Yaskawa INFORM job: DROP01.JBI

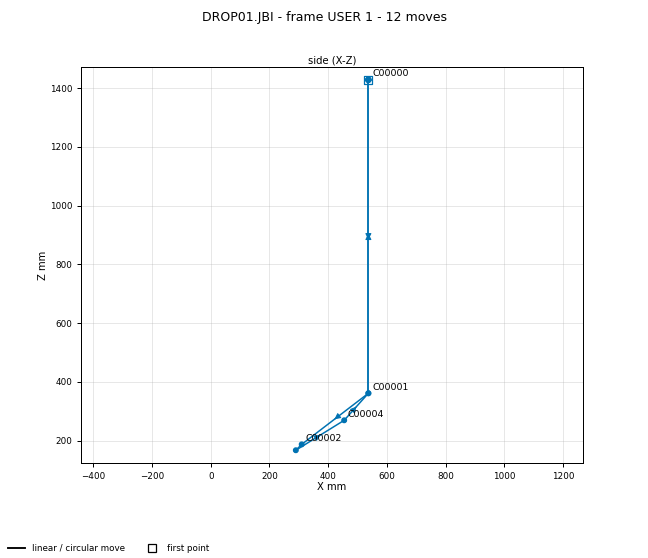
[picture p0: tool path of DROP01.JBI in frame USER 1, 12 of 12 moves have a stored position in this frame; points joined in program order, loops and branches not executed]
/JOB
//NAME DROP01
//POS
///NPOS 12,0,12,0,0,0
///USER 1
///TOOL 0
///POSTYPE USER
///RECTAN
///RCONF 0,0,0,0,0,0,0,0,0,0,0,0,0,0,0,0,0,0,0,0,0,0,0,0
C00000=536.880,595.000,1428.000,180.0000,0.0000,0.0000
C00001=536.880,595.000,360.810,180.0000,0.0000,0.0000
C00002=309.800,595.000,186.810,180.0000,0.0000,0.0000
C00003=289.800,595.000,166.810,180.0000,0.0000,0.0000
C00004=454.520,595.000,268.810,180.0000,0.0000,0.0000
C00005=536.880,595.000,360.810,180.0000,0.0000,0.0000
C00006=536.880,595.000,1428.000,180.0000,0.0000,0.0000
C00007=536.880,595.000,1428.000,180.0000,0.0000,0.0000
C00008=536.880,595.000,1428.000,180.0000,0.0000,0.0000
C00009=536.880,595.000,1428.000,180.0000,0.0000,0.0000
C00010=536.880,595.000,1428.000,180.0000,0.0000,0.0000
C00011=536.880,595.000,1428.000,180.0000,0.0000,0.0000
///POSTYPE PULSE
///PULSE
EC00000=359
EC00001=359
EC00002=359
EC00003=359
EC00004=359
EC00005=359
EC00006=359
EC00007=359
EC00008=359
EC00009=359
EC00010=359
EC00011=359
//INST
///DATE 2017/03/23 14:39
///ATTR SC,RW,RJ
////FRAME USER 1
///GROUP1 RB1,ST1
NOP
MOVL C00000 EC00000 V=1600.0
MOVL C00001 EC00001 V=1600.0
MOVL C00002 EC00002 V=1600.0
CALL JOB:GRIPERONOFF
MOVL C00003 EC00003 V=1600.0
MOVL C00004 EC00004 V=1600.0
MOVL C00005 EC00005 V=1600.0
MOVL C00006 EC00006 V=1600.0
MOVL C00007 EC00007 V=1600.0
MOVL C00008 EC00008 V=1600.0
MOVL C00009 EC00009 V=1600.0
MOVL C00010 EC00010 V=1600.0
MOVL C00011 EC00011 V=1600.0
END
